KUKA KRL data list: KVP_SendRelPos.dat

&ACCESS RVO
&REL 3
DEFDAT KVP_SendRelPos PUBLIC

DECL E6POS MyRelPos
DECL BOOL MyRelBool

ENDDAT
